(* PLC project testLD.project, CODESYS CODESYS V3.5 SP10 *)
(* stored: creationDateTime 2018-02-21T15:24:54.8270094, modificationDateTime 2018-02-21T15:24:46.3235105 *)

PROGRAM POU
  VAR
    n1 : BOOL;
    n2 : BOOL;
    n3 : BOOL;
    n4 : BOOL;
    n5 : BOOL;
    n6 : BOOL;
    n7 : BOOL;
    n8 : BOOL;
    n9 : BOOL;
    n10 : BOOL;
    n11 : BOOL;
    n12 : BOOL;
    n13 : BOOL;
    n14 : BOOL;
    n15 : BOOL;
  END_VAR

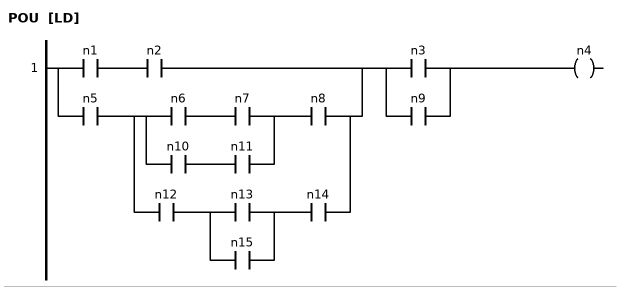
(* LD diagram, written out as Structured Text *)
n4 := (n1 AND n2 OR n5 AND (n6 AND n7 OR n10 AND n11) AND n8 OR n5 AND n12 AND (n13 OR n15) AND n14) AND (n3 OR n9);
END_PROGRAM

CONFIGURATION Application
  RESOURCE Application ON PLC
    TASK Task(INTERVAL := T#20ms, PRIORITY := 1);
    PROGRAM POU WITH Task : POU;
  END_RESOURCE
END_CONFIGURATION
